(* CoDeSys 2.3 export: DMX.EXP *)

(* POU DMX, FBD *)
PROGRAM DMX
VAR
	DMX_Master				: FbDMX_StageProfi;
		Enable				: BOOL := TRUE ;
		PortNumber			: WORD := 10001;
		FirstChannel		: WORD := 1;
		NumberOfChannels	: BYTE := 255;
		Ready				: BOOL;
		Connect				: BOOL;
		ErrorCode			: DINT;
		ErrorWatchdog		: BOOL;
END_VAR
VAR_INPUT RETAIN
		IPaddress			: STRING(16) := '192.168.1.120';
END_VAR
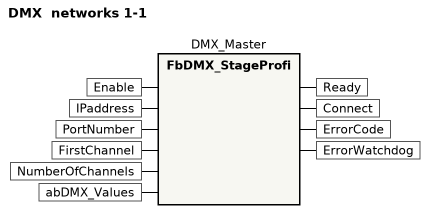
_FBD_ (* Function Block Diagram *)
NETWORK 1
	DMX_Master:FbDMX_StageProfi(Enable, IPaddress, PortNumber, FirstChannel, NumberOfChannels, abDMX_Values, out 2 => Connect, out 3 => ErrorCode, out 4 => ErrorWatchdog) => Ready
_END_FBD_
END_PROGRAM
